FUNCTION_BLOCK IMAGE_SAVER
  {SET_ATTRIBUTE(OpcUa, SERVICE)}
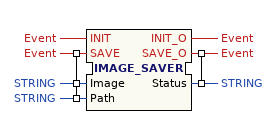
  EVENT_INPUT
    INIT;
    SAVE WITH Image, Path;
  END_EVENT
  EVENT_OUTPUT
    INIT_O;
    SAVE_O WITH Status;
  END_EVENT
  VAR_INPUT
    Image : STRING; (* Encoded image *)
    Path : STRING;
  END_VAR
  VAR_OUTPUT
    Status : STRING;
  END_VAR
END_FUNCTION_BLOCK
